FUNCTION_BLOCK Controller (* Composite Function Block Type *)
  (* Standard: 61499-2 *)
  (* Version 0.0, 7/13/2016, Andrei, nxtControl GmbH, template *)
  PACKAGE Main;
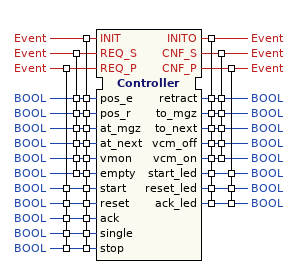
  EVENT_INPUT
    INIT WITH pos_e, pos_r, at_mgz, at_next, vmon, empty, start, reset, ack, single, stop; (* Initialization Request *)
    REQ_S WITH pos_e, pos_r, at_mgz, at_next, vmon, empty; (* Normal Execution Request *)
    REQ_P WITH start, reset, ack, single, stop;
  END_EVENT
  EVENT_OUTPUT
    INITO WITH retract, to_mgz, to_next, vcm_off, vcm_on, start_led, reset_led, ack_led; (* Initialization Confirm *)
    CNF_S WITH retract, to_mgz, to_next, vcm_off, vcm_on; (* Execution Confirmation *)
    CNF_P WITH start_led, reset_led, ack_led;
  END_EVENT
  VAR_INPUT
    pos_e : BOOL; (* Input event qualifier *)
    pos_r : BOOL;
    at_mgz : BOOL;
    at_next : BOOL;
    vmon : BOOL;
    empty : BOOL;
    start : BOOL;
    reset : BOOL;
    ack : BOOL;
    single : BOOL;
    stop : BOOL;
  END_VAR
  VAR_OUTPUT
    retract : BOOL; (* Output event qualifier *)
    to_mgz : BOOL;
    to_next : BOOL;
    vcm_off : BOOL;
    vcm_on : BOOL;
    start_led : BOOL;
    reset_led : BOOL;
    ack_led : BOOL;
  END_VAR
END_FUNCTION_BLOCK
